Yaskawa INFORM job: BUNNY.JBI

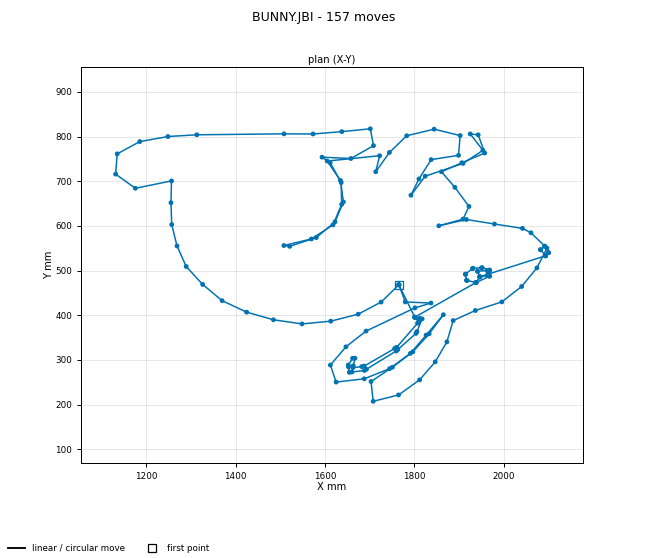
[picture p0: tool path of BUNNY.JBI, 157 of 157 moves have a stored position in this frame; points joined in program order, loops and branches not executed]
/JOB
//NAME BUNNY
//POS
///NPOS 157,0,0,0
///TOOL 0
///RECTAN
///RCONF 0,0,0,0,0
C000=1765.304,468.211,14.730,-176.06,5.36,66.50
C001=1765.304,468.211,14.730,-176.06,5.36,66.50
C002=1725.514,429.482,14.730,-176.06,5.36,66.50
C003=1674.181,402.379,14.730,-176.06,5.36,66.50
C004=1612.803,386.733,14.730,-176.06,5.36,66.50
C005=1548.342,380.581,14.730,-176.06,5.36,66.50
C006=1484.445,389.856,14.730,-176.06,5.36,66.50
C007=1424.419,406.956,14.730,-176.06,5.36,66.50
C008=1369.375,432.624,14.730,-176.06,5.36,66.50
C009=1325.842,469.004,14.730,-176.06,5.36,66.50
C010=1289.041,509.165,14.730,-176.06,5.36,66.50
C011=1268.473,555.189,14.730,-176.06,5.36,66.50
C012=1256.643,603.044,14.730,-176.06,5.36,66.50
C013=1254.908,651.971,14.730,-176.06,5.36,66.50
C014=1256.172,700.811,14.730,-176.06,5.36,66.50
C015=1175.163,684.371,14.730,-176.06,5.36,66.50
C016=1131.024,716.046,14.730,-176.06,5.36,66.50
C017=1134.541,761.399,14.730,-176.06,5.36,66.50
C018=1185.080,788.877,14.730,-176.06,5.36,66.50
C019=1248.113,800.199,14.730,-176.06,5.36,66.50
C020=1312.889,804.127,14.730,-176.06,5.36,66.50
C021=1508.003,806.212,14.730,-176.06,5.36,66.50
C022=1573.073,805.911,14.730,-176.06,5.36,66.50
C023=1637.486,811.150,14.730,-176.06,5.36,66.50
C024=1701.376,817.538,14.730,-176.06,5.36,66.50
C025=1708.487,779.779,14.730,-176.06,5.36,66.50
C026=1657.889,750.977,14.730,-176.06,5.36,66.50
C027=1593.251,753.973,14.730,-176.06,5.36,66.50
C028=1611.479,741.653,14.730,-176.06,5.36,66.50
C029=1636.173,697.045,14.730,-176.06,5.36,66.50
C030=1637.177,648.357,14.730,-176.06,5.36,66.50
C031=1617.890,602.528,14.730,-176.06,5.36,66.50
C032=1569.380,570.789,14.730,-176.06,5.36,66.50
C033=1507.760,556.170,14.730,-176.06,5.36,66.50
C034=1520.698,554.285,14.730,-176.06,5.36,66.50
C035=1580.317,573.903,14.730,-176.06,5.36,66.50
C036=1622.348,609.213,14.730,-176.06,5.36,66.50
C037=1641.048,653.799,14.730,-176.06,5.36,66.50
C038=1634.483,701.740,14.730,-176.06,5.36,66.50
C039=1604.817,745.303,14.730,-176.06,5.36,66.50
C040=1722.231,757.250,14.730,-176.06,5.36,66.50
C041=1713.489,721.393,14.730,-176.06,5.36,66.50
C042=1744.151,764.481,14.730,-176.06,5.36,66.50
C043=1782.896,801.964,14.730,-176.06,5.36,66.50
C044=1844.189,816.675,14.730,-176.06,5.36,66.50
C045=1902.534,802.378,14.730,-176.06,5.36,66.50
C046=1898.876,758.087,14.730,-176.06,5.36,66.50
C047=1837.593,748.477,14.730,-176.06,5.36,66.50
C048=1810.266,705.304,14.730,-176.06,5.36,66.50
C049=1792.296,668.763,14.730,-176.06,5.36,66.50
C050=1824.269,711.392,14.730,-176.06,5.36,66.50
C051=1909.078,740.055,14.730,-176.06,5.36,66.50
C052=1953.532,769.361,14.730,-176.06,5.36,66.50
C053=1925.198,806.010,14.730,-176.06,5.36,66.50
C054=1942.946,804.019,14.730,-176.06,5.36,66.50
C055=1957.614,763.273,14.730,-176.06,5.36,66.50
C056=1906.483,741.578,14.730,-176.06,5.36,66.50
C057=1860.641,721.315,14.730,-176.06,5.36,66.50
C058=1890.725,686.443,14.730,-176.06,5.36,66.50
C059=1922.328,643.659,14.730,-176.06,5.36,66.50
C060=1908.846,615.173,14.730,-176.06,5.36,66.50
C061=1854.764,600.264,14.730,-176.06,5.36,66.50
C062=1916.448,614.419,14.730,-176.06,5.36,66.50
C063=1979.253,604.308,14.730,-176.06,5.36,66.50
C064=2042.114,594.507,14.730,-176.06,5.36,66.50
C065=2061.109,584.635,14.730,-176.06,5.36,66.50
C066=2096.957,550.229,14.730,-176.06,5.36,66.50
C067=2074.408,506.016,14.730,-176.06,5.36,66.50
C068=2040.216,464.382,14.730,-176.06,5.36,66.50
C069=1995.858,429.910,14.730,-176.06,5.36,66.50
C070=1936.650,410.655,14.730,-176.06,5.36,66.50
C071=1886.920,388.098,14.730,-176.06,5.36,66.50
C072=1872.803,340.319,14.730,-176.06,5.36,66.50
C073=1846.718,295.696,14.730,-176.06,5.36,66.50
C074=1811.697,255.264,14.730,-176.06,5.36,66.50
C075=1764.600,221.489,14.730,-176.06,5.36,66.50
C076=1707.782,207.277,14.730,-176.06,5.36,66.50
C077=1703.010,251.623,14.730,-176.06,5.36,66.50
C078=1750.792,283.590,14.730,-176.06,5.36,66.50
C079=1796.687,318.190,14.730,-176.06,5.36,66.50
C080=1833.203,358.463,14.730,-176.06,5.36,66.50
C081=1864.991,401.171,14.730,-176.06,5.36,66.50
C082=1826.273,355.436,14.730,-176.06,5.36,66.50
C083=1791.132,314.546,14.730,-176.06,5.36,66.50
C084=1744.508,280.402,14.730,-176.06,5.36,66.50
C085=1687.772,257.682,14.730,-176.06,5.36,66.50
C086=1624.815,250.357,14.730,-176.06,5.36,66.50
C087=1611.891,288.399,14.730,-176.06,5.36,66.50
C088=1646.768,329.305,14.730,-176.06,5.36,66.50
C089=1691.852,364.559,14.730,-176.06,5.36,66.50
C090=1801.341,416.607,14.730,-176.06,5.36,66.50
C091=1837.216,427.292,14.730,-176.06,5.36,66.50
C092=1779.569,429.754,14.730,-176.06,5.36,66.50
C093=1765.304,468.211,14.730,-176.06,5.36,66.50
C094=1765.304,468.211,14.730,-176.06,5.36,66.50
C095=1800.873,395.599,14.730,-176.06,5.36,66.50
C096=1800.873,395.599,14.730,-176.06,5.36,66.50
C097=1811.854,393.121,14.730,-176.06,5.36,66.50
C098=1817.344,391.882,14.730,-176.06,5.36,66.50
C099=1805.729,363.381,14.730,-176.06,5.36,66.50
C100=1803.671,359.405,14.730,-176.06,5.36,66.50
C101=1763.008,323.158,14.730,-176.06,5.36,66.50
C102=1759.311,319.863,14.730,-176.06,5.36,66.50
C103=1692.640,279.049,14.730,-176.06,5.36,66.50
C104=1688.185,276.336,14.730,-176.06,5.36,66.50
C105=1660.056,272.769,14.730,-176.06,5.36,66.50
C106=1654.387,272.129,14.730,-176.06,5.36,66.50
C107=1652.498,284.279,14.730,-176.06,5.36,66.50
C108=1652.141,288.582,14.730,-176.06,5.36,66.50
C109=1661.710,303.568,14.730,-176.06,5.36,66.50
C110=1667.041,303.763,14.730,-176.06,5.36,66.50
C111=1663.271,286.752,14.730,-176.06,5.36,66.50
C112=1662.329,282.499,14.730,-176.06,5.36,66.50
C113=1682.120,284.987,14.730,-176.06,5.36,66.50
C114=1687.611,286.171,14.730,-176.06,5.36,66.50
C115=1755.824,325.544,14.730,-176.06,5.36,66.50
C116=1760.333,328.197,14.730,-176.06,5.36,66.50
C117=1807.208,382.199,14.730,-176.06,5.36,66.50
C118=1809.772,386.055,14.730,-176.06,5.36,66.50
C119=1800.873,395.599,14.730,-176.06,5.36,66.50
C120=1800.873,395.599,14.730,-176.06,5.36,66.50
C121=1938.066,473.306,14.730,-176.06,5.36,66.50
C122=1938.066,473.306,14.730,-176.06,5.36,66.50
C123=1918.149,477.916,14.730,-176.06,5.36,66.50
C124=1916.617,478.270,14.730,-176.06,5.36,66.50
C125=1914.505,491.164,14.730,-176.06,5.36,66.50
C126=1914.360,492.364,14.730,-176.06,5.36,66.50
C127=1930.175,504.314,14.730,-176.06,5.36,66.50
C128=1931.316,505.155,14.730,-176.06,5.36,66.50
C129=1950.485,506.357,14.730,-176.06,5.36,66.50
C130=1952.051,506.297,14.730,-176.06,5.36,66.50
C131=1968.423,501.371,14.730,-176.06,5.36,66.50
C132=1968.554,500.233,14.730,-176.06,5.36,66.50
C133=1968.554,488.176,14.730,-176.06,5.36,66.50
C134=1968.158,487.137,14.730,-176.06,5.36,66.50
C135=1938.066,473.306,14.730,-176.06,5.36,66.50
C136=1938.066,473.306,14.730,-176.06,5.36,66.50
C137=1946.535,486.045,14.730,-176.06,5.36,66.50
C138=1946.535,486.045,14.730,-176.06,5.36,66.50
C139=1941.710,498.143,14.730,-176.06,5.36,66.50
C140=1941.500,498.669,14.730,-176.06,5.36,66.50
C141=1963.134,500.039,14.730,-176.06,5.36,66.50
C142=1963.473,499.764,14.730,-176.06,5.36,66.50
C143=1963.473,489.331,14.730,-176.06,5.36,66.50
C144=1963.473,488.781,14.730,-176.06,5.36,66.50
C145=1946.535,486.045,14.730,-176.06,5.36,66.50
C146=1946.535,486.045,14.730,-176.06,5.36,66.50
C147=2093.892,533.179,14.730,-176.06,5.36,66.50
C148=2093.892,533.179,14.730,-176.06,5.36,66.50
C149=2082.614,546.508,14.730,-176.06,5.36,66.50
C150=2082.238,546.953,14.730,-176.06,5.36,66.50
C151=2091.671,554.439,14.730,-176.06,5.36,66.50
C152=2092.166,554.811,14.730,-176.06,5.36,66.50
C153=2100.260,540.283,14.730,-176.06,5.36,66.50
C154=2100.529,539.797,14.730,-176.06,5.36,66.50
C155=2093.892,533.179,14.730,-176.06,5.36,66.50
C156=2093.892,533.179,14.730,-176.06,5.36,66.50
//INST
///DATE 2014/11/08 20:23
///ATTR 0,0,0,0,0,0,0,0,0,0,0,0,1,1,0,0
///FRAME BASE
NOP
*1
MOVL C000 V=200.0 CONT
PAUSE
MOVL C001 V=200.0 CONT
MOVL C002 V=200.0 CONT
MOVL C003 V=200.0 CONT
MOVL C004 V=200.0 CONT
MOVL C005 V=200.0 CONT
MOVL C006 V=200.0 CONT
MOVL C007 V=200.0 CONT
MOVL C008 V=200.0 CONT
MOVL C009 V=200.0 CONT
MOVL C010 V=200.0 CONT
MOVL C011 V=200.0 CONT
MOVL C012 V=200.0 CONT
MOVL C013 V=200.0 CONT
MOVL C014 V=200.0 CONT
MOVL C015 V=200.0 CONT
MOVL C016 V=200.0 CONT
MOVL C017 V=200.0 CONT
MOVL C018 V=200.0 CONT
MOVL C019 V=200.0 CONT
MOVL C020 V=200.0 CONT
MOVL C021 V=200.0 CONT
MOVL C022 V=200.0 CONT
MOVL C023 V=200.0 CONT
MOVL C024 V=200.0 CONT
MOVL C025 V=200.0 CONT
MOVL C026 V=200.0 CONT
MOVL C027 V=200.0 CONT
MOVL C028 V=200.0 CONT
MOVL C029 V=200.0 CONT
MOVL C030 V=200.0 CONT
MOVL C031 V=200.0 CONT
MOVL C032 V=200.0 CONT
MOVL C033 V=200.0 CONT
MOVL C034 V=200.0 CONT
MOVL C035 V=200.0 CONT
MOVL C036 V=200.0 CONT
MOVL C037 V=200.0 CONT
MOVL C038 V=200.0 CONT
MOVL C039 V=200.0 CONT
MOVL C040 V=200.0 CONT
MOVL C041 V=200.0 CONT
MOVL C042 V=200.0 CONT
MOVL C043 V=200.0 CONT
MOVL C044 V=200.0 CONT
MOVL C045 V=200.0 CONT
MOVL C046 V=200.0 CONT
MOVL C047 V=200.0 CONT
MOVL C048 V=200.0 CONT
MOVL C049 V=200.0 CONT
MOVL C050 V=200.0 CONT
MOVL C051 V=200.0 CONT
MOVL C052 V=200.0 CONT
MOVL C053 V=200.0 CONT
MOVL C054 V=200.0 CONT
MOVL C055 V=200.0 CONT
MOVL C056 V=200.0 CONT
MOVL C057 V=200.0 CONT
MOVL C058 V=200.0 CONT
MOVL C059 V=200.0 CONT
MOVL C060 V=200.0 CONT
MOVL C061 V=200.0 CONT
MOVL C062 V=200.0 CONT
MOVL C063 V=200.0 CONT
MOVL C064 V=200.0 CONT
MOVL C065 V=200.0 CONT
MOVL C066 V=200.0 CONT
MOVL C067 V=200.0 CONT
MOVL C068 V=200.0 CONT
MOVL C069 V=200.0 CONT
MOVL C070 V=200.0 CONT
MOVL C071 V=200.0 CONT
MOVL C072 V=200.0 CONT
MOVL C073 V=200.0 CONT
MOVL C074 V=200.0 CONT
MOVL C075 V=200.0 CONT
MOVL C076 V=200.0 CONT
MOVL C077 V=200.0 CONT
MOVL C078 V=200.0 CONT
MOVL C079 V=200.0 CONT
MOVL C080 V=200.0 CONT
MOVL C081 V=200.0 CONT
MOVL C082 V=200.0 CONT
MOVL C083 V=200.0 CONT
MOVL C084 V=200.0 CONT
MOVL C085 V=200.0 CONT
MOVL C086 V=200.0 CONT
MOVL C087 V=200.0 CONT
MOVL C088 V=200.0 CONT
MOVL C089 V=200.0 CONT
MOVL C090 V=200.0 CONT
MOVL C091 V=200.0 CONT
MOVL C092 V=200.0 CONT
MOVL C093 V=200.0 CONT
MOVL C094 V=200.0 CONT
MOVL C095 V=200.0 CONT
MOVL C096 V=200.0 CONT
MOVL C097 V=200.0 CONT
MOVL C098 V=200.0 CONT
MOVL C099 V=200.0 CONT
MOVL C100 V=200.0 CONT
MOVL C101 V=200.0 CONT
MOVL C102 V=200.0 CONT
MOVL C103 V=200.0 CONT
MOVL C104 V=200.0 CONT
MOVL C105 V=200.0 CONT
MOVL C106 V=200.0 CONT
MOVL C107 V=200.0 CONT
MOVL C108 V=200.0 CONT
MOVL C109 V=200.0 CONT
MOVL C110 V=200.0 CONT
MOVL C111 V=200.0 CONT
MOVL C112 V=200.0 CONT
MOVL C113 V=200.0 CONT
MOVL C114 V=200.0 CONT
MOVL C115 V=200.0 CONT
MOVL C116 V=200.0 CONT
MOVL C117 V=200.0 CONT
MOVL C118 V=200.0 CONT
MOVL C119 V=200.0 CONT
MOVL C120 V=200.0 CONT
MOVL C121 V=200.0 CONT
MOVL C122 V=200.0 CONT
MOVL C123 V=200.0 CONT
MOVL C124 V=200.0 CONT
MOVL C125 V=200.0 CONT
MOVL C126 V=200.0 CONT
MOVL C127 V=200.0 CONT
MOVL C128 V=200.0 CONT
MOVL C129 V=200.0 CONT
MOVL C130 V=200.0 CONT
MOVL C131 V=200.0 CONT
MOVL C132 V=200.0 CONT
MOVL C133 V=200.0 CONT
MOVL C134 V=200.0 CONT
MOVL C135 V=200.0 CONT
MOVL C136 V=200.0 CONT
MOVL C137 V=200.0 CONT
MOVL C138 V=200.0 CONT
MOVL C139 V=200.0 CONT
MOVL C140 V=200.0 CONT
MOVL C141 V=200.0 CONT
MOVL C142 V=200.0 CONT
MOVL C143 V=200.0 CONT
MOVL C144 V=200.0 CONT
MOVL C145 V=200.0 CONT
MOVL C146 V=200.0 CONT
MOVL C147 V=200.0 CONT
MOVL C148 V=200.0 CONT
MOVL C149 V=200.0 CONT
MOVL C150 V=200.0 CONT
MOVL C151 V=200.0 CONT
MOVL C152 V=200.0 CONT
MOVL C153 V=200.0 CONT
MOVL C154 V=200.0 CONT
MOVL C155 V=200.0 CONT
MOVL C156 V=200.0 CONT
JUMP *1
END
